{attribute 'linkalways'} 
{attribute 'no_explicit_call' := 'This FB is a CLASS and must be accessed using methods or properties'}
{attribute 'enable_dynamic_creation'}
FUNCTION_BLOCK _ETcVnDiffusivityTypeKAZE EXTENDS EnumDatatypeBase
VAR
	localData : ETcVnDiffusivityTypeKAZE;
	activeData : REFERENCE TO ETcVnDiffusivityTypeKAZE;
	enumBaseDatatype : _DINT(localData);
END_VAR

METHOD PRIVATE AddLocalEnumeration
VAR_INPUT
	Enumeration : T_MAXSTRING;
	Value : ETcVnDiffusivityTypeKAZE;
END_VAR
AddEnumeration(Enumeration, Value);
END_METHOD

PROPERTY PUBLIC Address : PVOID
GET
Address := ADR(activeData);
END_GET
END_PROPERTY

METHOD PUBLIC ClearReference
VAR_INPUT
END_VAR
activeData REF= localData;
SetBaseDatatypeReference();
END_METHOD

METHOD PUBLIC Clone : I_Datatype
VAR
    pClone : POINTER TO _ETcVnDiffusivityTypeKAZE;
END_VAR
pClone := __NEW(_ETcVnDiffusivityTypeKAZE(InitialValue := Value));
Clone := pClone^;
END_METHOD

METHOD FB_init : BOOL
VAR_INPUT
	bInitRetains : BOOL; // if TRUE, the retain variables are initialized (warm start / cold start)
	bInCopyCode : BOOL;  // if TRUE, the instance afterwards gets moved into the copy code (online change)
	InitialValue : ETcVnDiffusivityTypeKAZE;
END_VAR
localData := InitialValue;
AddBaseDatatype(enumBaseDatatype);
ClearReference();

AddLocalEnumeration('TCVN_DT1_KAZE_PM_G1', ETcVnDiffusivityTypeKAZE.TCVN_DT1_KAZE_PM_G1);
AddLocalEnumeration('TCVN_DT1_KAZE_PM_G2', ETcVnDiffusivityTypeKAZE.TCVN_DT1_KAZE_PM_G2);
AddLocalEnumeration('TCVN_DT1_KAZE_WEICKERT', ETcVnDiffusivityTypeKAZE.TCVN_DT1_KAZE_WEICKERT);
AddLocalEnumeration('TCVN_DT1_KAZE_CHARBONNIER', ETcVnDiffusivityTypeKAZE.TCVN_DT1_KAZE_CHARBONNIER);
END_METHOD

PROPERTY PUBLIC Identifier : T_MAXSTRING
GET
Identifier := 'ETcVnDiffusivityTypeKAZE';
END_GET
END_PROPERTY

METHOD IsEnumeratorValueEqual : BOOL
VAR_INPUT
	Enumerator : I_KeyValueForwardEnumerator;
END_VAR
VAR
	storedValue : ETcVnDiffusivityTypeKAZE;
END_VAR
IF NOT Enumerator.TryGet(storedValue) THEN
	RETURN;
END_IF

IsEnumeratorValueEqual := storedValue = activeData;
END_METHOD

METHOD PUBLIC MakeReferenceTo
VAR_INPUT
	ReferenceTarget : REFERENCE TO ETcVnDiffusivityTypeKAZE;
END_VAR
activeData REF= ReferenceTarget;
SetBaseDatatypeReference();
END_METHOD

METHOD PROTECTED SetBaseDatatypeReference
VAR_INPUT
END_VAR
enumBaseDatatype.MakeReferenceTo(activeData);
END_METHOD

PROPERTY PUBLIC Size : UDINT
GET
Size := SIZEOF(activeData);
END_GET
END_PROPERTY

METHOD TryMakeReferenceTo : BOOL
VAR_INPUT
	Target : I_Datatype;
END_VAR
VAR
	targetAsEnum : I_EnumDatatype;
	pTargetData : POINTER TO ETcVnDiffusivityTypeKAZE;
END_VAR
IF NOT Target.TryResolveAsEnumDatatype(targetAsEnum) THEN
	RETURN;
END_IF

IF targetAsEnum.Identifier <> Identifier THEN
	RETURN;
END_IF

pTargetData := Target.Address;
activeData REF= pTargetData^;
SetBaseDatatypeReference();
TryMakeReferenceTo := TRUE;
END_METHOD

PROPERTY PUBLIC Value : ETcVnDiffusivityTypeKAZE
GET
Value := activeData;
END_GET
SET
activeData := Value;
END_SET
END_PROPERTY

END_FUNCTION_BLOCK

(* stored: Version 1.1.0.1, ProductVersion 3.1.4024.12
   POU _ETcVnDiffusivityTypeKAZE: Id {de3c724f-c8b2-47c1-8eef-2eb1b41c5821}, SpecialFunc None
   Folder Constructor: Id {d03ed285-64c9-4e98-8e42-6b10856a48f1}
   Folder Private: Id {ffabc81c-1f05-4024-8053-599571fc6dd5}
   Folder Protected: Id {a86c97cb-48f8-4859-8994-008013a916b6}
   Method AddLocalEnumeration: Id {83369ed4-b32a-4ce4-a928-5a82cc7323f2}
   Property Address: Id {352855b2-30c1-4691-9ea3-3a32df8aa674}
   Get Get: Id {19eaf390-fa16-465c-aa09-6a5798f3fbc3}
   Method ClearReference: Id {1fcb9a7c-6903-4648-b010-dcc24250ceee}
   Method Clone: Id {7dab210d-759a-4397-81e4-befa4ef4e974}
   Method FB_init: Id {227b4b11-b1ef-47fc-b8c4-2c50934502f2}
   Property Identifier: Id {439fadb6-e9fc-4836-93dc-a516e071f152}
   Get Get: Id {f3eac933-a1d1-4842-a53f-80f35064a529}
   Method IsEnumeratorValueEqual: Id {acb0921a-d560-4752-b3aa-86060bd6b061}
   Method MakeReferenceTo: Id {854c40fe-ec91-4b12-bb01-079ddb92026a}
   Method SetBaseDatatypeReference: Id {838f5702-c3fe-4f3d-9712-6882800b5b4b}
   Property Size: Id {9318f610-d64d-4d4f-babc-287e9fa19050}
   Get Get: Id {bba2e89b-5e19-4e02-974e-363c1c63794f}
   Method TryMakeReferenceTo: Id {266ca28d-2b81-4152-92ec-bea3e3c949a7}
   Property Value: Id {a5b92b6a-a54a-4ad8-b305-50a3d58ff3a2}
   Get Get: Id {603ba6f7-d67e-4dbb-90ad-a334093bdc91}
   Set Set: Id {5b88df2b-ec40-46f2-86ae-d424bec03f4b} *)
